RoboDK station: Botellas.rdk

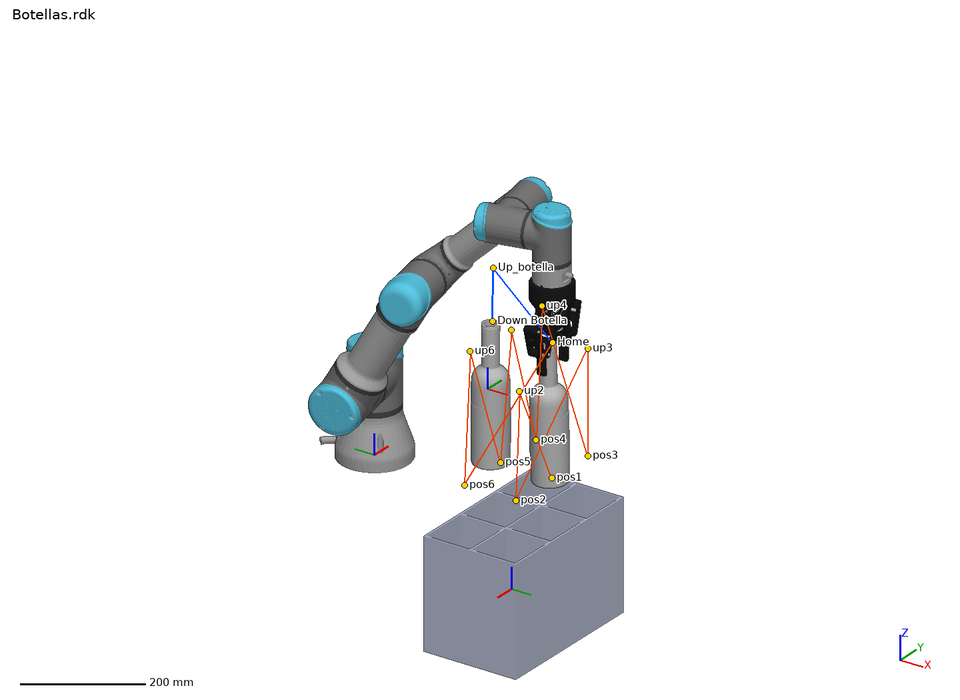
[picture v0: the station drawn from its stored meshes, robots at their saved joint values, targets as dots, program paths as lines]
Station Botellas (saved by RoboDK 5.5.1). Poses are relative to the parent item; angles as X-Y-Z fixed-axis rotations.
  - frame General_Frame at (0, 0, 0) mm
    - frame Basked_frame at (207.27, -229.59, -204.34) mm, rotated rx 0 ry 0 rz -90 deg
      - object basked at (110, 100, 0) mm, rotated rx 90 ry 0 rz 0 deg, size 299.8 x 204 x 180 mm, geometry from basked.STEP
      - target Home (Cartesian target) at (110.35, 156.78, 524.07) mm, rotated rx -179.23 ry -0.45 rz 2.88 deg; joints [66.707, -44.377, -17.878, -28.633, -90.069, -26.01] of UR3
      - target Up_botella (Cartesian target) at (-237.12, -202.06, 416.73) mm, rotated rx -179.95 ry -1.36 rz 80.65 deg; joints [18.228, -102.65, -36.587, -131.35, 88.777, 27.749] of UR3
      - target Down Botella (Cartesian target) at (-237.39, -203.22, 322.06) mm, rotated rx -179.95 ry -1.36 rz 80.65 deg; joints [18.422, -91.283, -78.287, -101.02, 88.779, 27.943] of UR3
      - target pos1 (Cartesian target) at (113.59, 157.6, 285.25) mm, rotated rx -179.23 ry -0.45 rz 2.88 deg; joints [-79.433, -111.635, -98.244, -59.422, 89.448, 7.848] of UR3
      - target pos2 (Cartesian target) at (213.59, 157.6, 285.25) mm, rotated rx -179.23 ry -0.45 rz 2.88 deg; joints [-94.931, -116.793, -90.386, -62, 89.655, -7.65] of UR3
      - target pos3 (Cartesian target) at (13.59, 157.6, 285.25) mm, rotated rx -179.23 ry -0.45 rz 2.88 deg; joints [-64.241, -112.077, -97.509, -59.884, 89.284, 23.04] of UR3
      - target pos4 (Cartesian target) at (13.59, 57.6, 285.25) mm, rotated rx -179.23 ry -0.45 rz 2.88 deg; joints [-54.734, -89.561, -125.659, -54.376, 89.207, 32.548] of UR3
      - target pos5 (Cartesian target) at (113.59, 57.6, 285.25) mm, rotated rx -179.23 ry -0.45 rz 2.88 deg; joints [-75.265, -88.856, -126.471, -54.016, 89.399, 12.015] of UR3
      - target pos6 (Cartesian target) at (213.59, 57.6, 285.25) mm, rotated rx -179.23 ry -0.45 rz 2.88 deg; joints [-96.602, -96.663, -118.221, -54.285, 89.679, -9.32] of UR3
      - target up2 (Cartesian target) at (203.59, 157.6, 475.25) mm, rotated rx -179.24 ry -0.46 rz 2.87 deg; joints [-93.428, -114.816, -40.465, -113.916, 89.629, -6.133] of UR3
      - target up3 (Cartesian target) at (13.59, 157.6, 475.25) mm, rotated rx -179.23 ry -0.45 rz 2.88 deg; joints [-64.241, -109.05, -48.798, -111.622, 89.284, 23.04] of UR3
      - target up4 (Cartesian target) at (10.35, 66.78, 524.06) mm, rotated rx -179.22 ry -0.45 rz 2.9 deg; joints [-55.313, -90.927, -56.084, -122.568, 89.21, 31.954] of UR3
      - target up5 (Cartesian target) at (110.35, 76.78, 524.06) mm, rotated rx -179.23 ry -0.45 rz 2.88 deg; joints [-75.645, -92.413, -54.651, -122.275, 89.403, 11.635] of UR3
      - target up6 (Cartesian target) at (210.35, 66.78, 524.06) mm, rotated rx -179.23 ry -0.45 rz 2.88 deg; joints [43.008, -36.976, -48.838, -5.027, -89.706, -49.706] of UR3
      - object b5 at (-181.21, 133.26, 84.02) mm, rotated rx -117.73 ry -89.98 rz -91.75 deg, size 246.5 x 62 x 63.4 mm, geometry from b.stl
    - object b1 at (340.45, -48.38, -120.42) mm, rotated rx 0 ry -90 rz 60.52 deg, size 246.5 x 62 x 63.4 mm, geometry from b.stl
    - object b4 at (340.45, -48.38, -120.42) mm, rotated rx 0 ry -90 rz 60.52 deg, size 246.5 x 62 x 63.4 mm, geometry from b.stl
    - object b2 at (340.45, -48.38, -120.42) mm, rotated rx 0 ry -90 rz 60.52 deg, size 246.5 x 62 x 63.4 mm, geometry from b.stl
    - object b3 at (340.45, -48.38, -120.42) mm, rotated rx 0 ry -90 rz 60.52 deg, size 246.5 x 62 x 63.4 mm, geometry from b.stl
  - frame UR3 Base at (-10, -300, 0) mm, rotated rx 0 ry 0 rz 90.17 deg
    - robot UR3: 6 axes, payload 3 kg, reach 500 mm, repeatability 0.1 mm, weight 11 kg
        modified DH rows (alpha deg, a mm, theta deg, d mm): 0, 0, 0, 151.9; 90, 0, 180, 0; 0, 243.65, 0, 0; 0, 213, 0, 110.4; -90, 0, 0, 83.4; 90, 0, 180, 82.4
        joint limits [-360, -360, -360, -360, -360, -360] to [360, 360, 360, 360, 360, 360]; home [0, -90, -90, 0, 90, 0]; saved at [-78.898, -119.103, -17.513, -132.691, 89.442, 8.383]
      - tool RobotiQ 2F-85 Gripper (Closed), TCP at (0, 0, 130) mm, size 134.4 x 157.6 x 75 mm
        - object b6 at (335.49, 0.99, 225.93) mm, rotated rx -112.1 ry 88.68 rz -1.97 deg, size 246.5 x 62 x 63.4 mm, geometry from b.stl
      - tool RobotiQ 2F-85 Gripper (Open), TCP at (0, 0, 110) mm, size 147.4 x 146.8 x 75 mm
  - program Re-ubicar (9 instructions, listed below)
  - program pick_place (9 instructions, listed below)
  - program proceso (27 instructions, listed below)
  - program soltar (3 instructions, listed below)
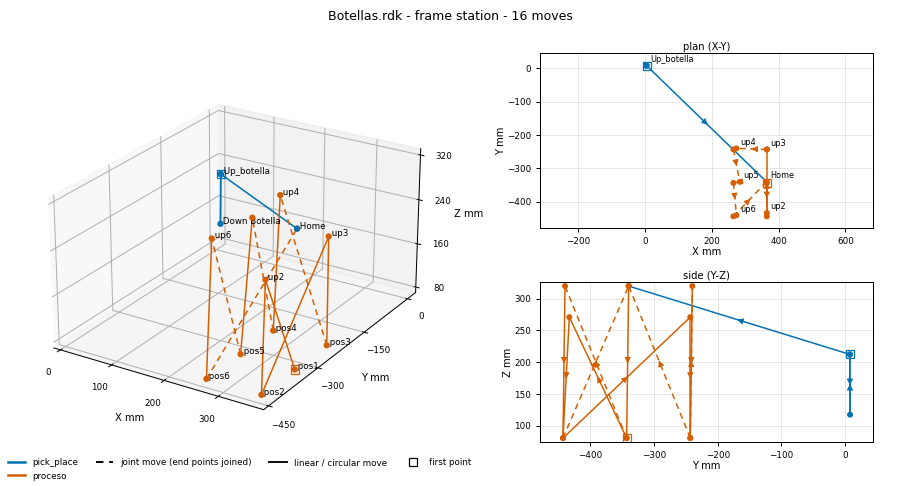
[picture p0: tool path of Botellas.rdk in frame station, 16 of 16 moves have a stored position in this frame; points joined in program order, loops and branches not executed]

--- program Re-ubicar (robot UR3) ---
  Reemplazar b1
  Reemplazar b4
  Reemplazar b2
  Reemplazar b3
  Reemplazar b5
  Reemplazar b6
  No definido
  Mostrar RobotiQ 2F-85 Gripper (Open)
  Ocultar RobotiQ 2F-85 Gripper (Closed)

--- program pick_place (robot UR3) ---
  Est. Ref.: Basked_frame
  Est. herr: RobotiQ 2F-85 Gripper (Open)
  MoveJ (Up_botella)
  MoveL (Down Botella)
  Mostrar RobotiQ 2F-85 Gripper (Closed)
  Ocultar RobotiQ 2F-85 Gripper (Open)
  Adjuntar a RobotiQ 2F-85 Gripper (Closed)
  MoveL (Up_botella)
  MoveL (Home)

--- program proceso (robot UR3) ---
  Est. Ref.: Basked_frame
  Est. herr: RobotiQ 2F-85 Gripper (Open)
  Llamar pick_place
  MoveL (pos1)
  Llamar soltar
  Llamar pick_place
  MoveL (Target 11) -> target up2
  MoveL (pos2)
  Llamar soltar
  Llamar pick_place
  MoveL (Target 11) -> target up3
  MoveL (pos3)
  Llamar soltar
  Llamar pick_place
  MoveJ (Target 12) -> target up4
  MoveL (pos4)
  Llamar soltar
  Llamar pick_place
  MoveJ (Target 13) -> target up5
  MoveL (pos5)
  Llamar soltar
  Llamar pick_place
  MoveJ (Target 15) -> target up6
  MoveL (pos6)
  Llamar soltar
  Llamar Program1
  MoveJ (Home)

--- program soltar (robot UR3) ---
  Separar de RobotiQ 2F-85 Gripper (Closed)
  Ocultar RobotiQ 2F-85 Gripper (Closed)
  Mostrar RobotiQ 2F-85 Gripper (Open)
